Fanuc KAREL source: kt00375.KL

PROGRAM KT00375
%NOLOCKGROUP
VAR
Y1 : ARRAY[2] OF BYTE
I2:INTEGER
OUT:BOOLEAN
BEGIN
Y1[1]=2
I2=3
OUT=(Y1[1] <=I2)
END KT00375
